% RSLogix 500 project Project_1.RSS, saved by version 8.30.00.16 %
PROJECT "UNTITLED"    % processor: Bul.1763 MicroLogix 1100 Series B %

PROGRAM FILES
  LAD 2 "MAIN"  3 rungs
  LAD 3 "DIGITAL IO"  5 rungs
  LAD 4 "CONTROL"  9 rungs

DATA FILES
  O0 OUTPUT  9 elements
  I1 INPUT  16 elements
  S2 STATUS  66 elements
  B3 BINARY  1 elements
  T4 TIMER  2 elements
  C5 COUNTER  1 elements
  R6 CONTROL  1 elements
  N7 INTEGER  1 elements
  F8 FLOAT  1 elements

LADDER 2 "MAIN"
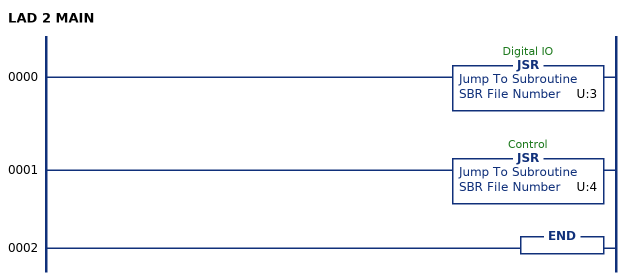
% Rung: 0 %
SOR JSR U:3 EOR
%   U:3  "Digital IO" %
% Rung: 1 %
SOR JSR U:4 EOR
%   U:4  "Control" %
% Rung: 2 %
SOR END EOR

LADDER 3 "DIGITAL IO"
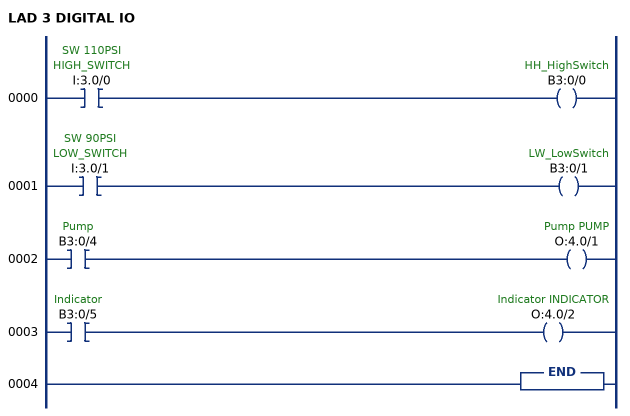
% Rung: 0 %
SOR XIC I:3.0/0 OTE B3:0/0 EOR
%   I:3.0/0  HIGH_SWITCH  "SW 110PSI" %
%   B3:0/0  "HH_HighSwitch" %
% Rung: 1 %
SOR XIC I:3.0/1 OTE B3:0/1 EOR
%   I:3.0/1  LOW_SWITCH  "SW 90PSI" %
%   B3:0/1  "LW_LowSwitch" %
% Rung: 2 %
SOR XIC B3:0/4 OTE O:4.0/1 EOR
%   B3:0/4  "Pump" %
%   O:4.0/1  PUMP  "Pump" %
% Rung: 3 %
SOR XIC B3:0/5 OTE O:4.0/2 EOR
%   B3:0/5  "Indicator" %
%   O:4.0/2  INDICATOR  "Indicator" %
% Rung: 4 %
SOR END EOR

LADDER 4 "CONTROL"
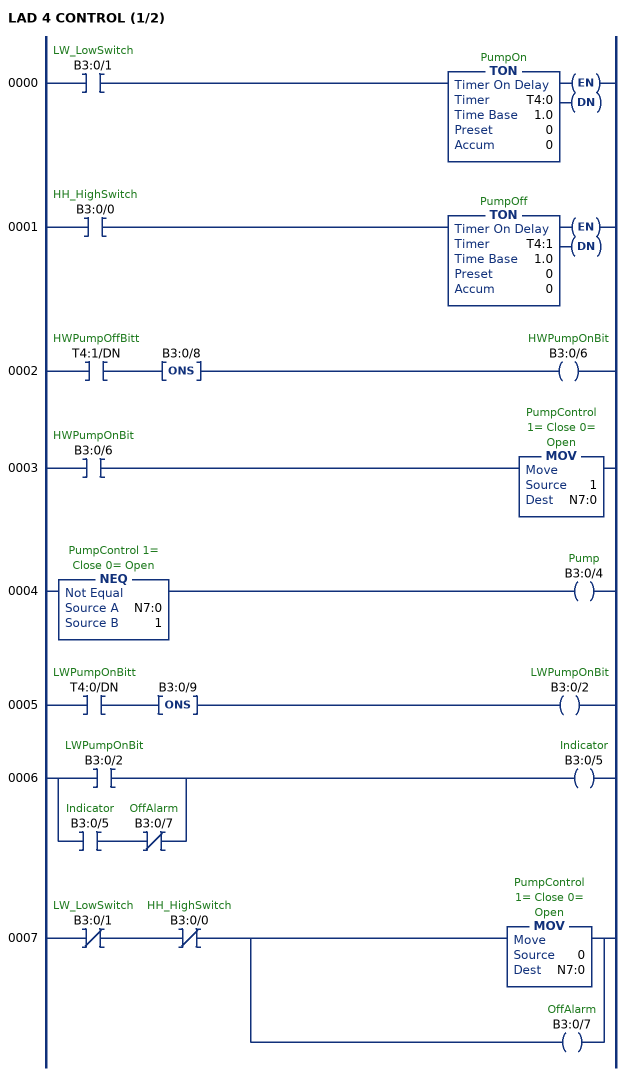
% Rung: 0 %
SOR XIC B3:0/1 TON T4:0 1.0 0 0 EOR
%   B3:0/1  "LW_LowSwitch" %
%   T4:0  "PumpOn" %
% Rung: 1 %
SOR XIC B3:0/0 TON T4:1 1.0 0 0 EOR
%   B3:0/0  "HH_HighSwitch" %
%   T4:1  "PumpOff" %
% Rung: 2 %
SOR XIC T4:1/DN ONS B3:0/8 OTE B3:0/6 EOR
%   T4:1/DN  "HWPumpOffBitt" %
%   B3:0/6  "HWPumpOnBit" %
% Rung: 3 %
SOR XIC B3:0/6 MOV 1 N7:0 EOR
%   B3:0/6  "HWPumpOnBit" %
%   N7:0  "PumpControl 1= Close 0= Open" %
% Rung: 4 %
SOR NEQ N7:0 1 OTE B3:0/4 EOR
%   N7:0  "PumpControl 1= Close 0= Open" %
%   B3:0/4  "Pump" %
% Rung: 5 %
SOR XIC T4:0/DN ONS B3:0/9 OTE B3:0/2 EOR
%   T4:0/DN  "LWPumpOnBitt" %
%   B3:0/2  "LWPumpOnBit" %
% Rung: 6 %
SOR BST XIC B3:0/2 NXB XIC B3:0/5 XIO B3:0/7 BND OTE B3:0/5 EOR
%   B3:0/2  "LWPumpOnBit" %
%   B3:0/5  "Indicator" %
%   B3:0/7  "OffAlarm" %
% Rung: 7 %
SOR XIO B3:0/1 XIO B3:0/0 BST MOV 0 N7:0 NXB OTE B3:0/7 BND EOR
%   B3:0/1  "LW_LowSwitch" %
%   B3:0/0  "HH_HighSwitch" %
%   N7:0  "PumpControl 1= Close 0= Open" %
%   B3:0/7  "OffAlarm" %

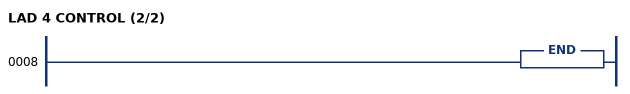
% Rung: 8 %
SOR END EOR

OTHER DOCUMENTED ADDRESSES
  B3:0/3  "Valve"
  O:4.0/0  VALVE  "Valve"
